REGION Network 51: UNIT 01 STATION 3 COAXIAL HIGH NUMBER OF DEAD PIXELS ALARM
   RUNG wire#powerrail
      { S7_Templates := "SrcType := Int" } EQ_Contact(in1 := "DB16002_U01_STA3_COAXIAL_CLIENT_INTERFACE".U1_STA3_CAM_Read.Variable.Status, in2 := -1)
      Contact( "DB16002_U01_STA3_COAXIAL_CLIENT_INTERFACE".U1_STA3_CAM_Read.Variable.FailedToConnectToCamera )
      wire#w1
      Contact( "DB7254_UNIT_01_STA_3_COAXIAL_ENABLE_DISABLE".ENABLED )
      wire#w2
      Coil( "DB16000_OPC_UA_TRIGGER_ALARM".CLIENT.U1_STA3_COAXIAL.ALARMS.HIGH_NUM_DEAD_PIXELS_A )
   END_RUNG
   RUNG wire#powerrail
      Contact( "DB16000_OPC_UA_TRIGGER_ALARM".CLIENT.U1_STA3_COAXIAL.ALARMS.HIGH_NUM_DEAD_PIXELS_A )
      I_Contact( "DB2120_MPP_ITC_IPC".RESET_FAULTS )
   END_RUNG wire#w1
   RUNG wire#w2
      Coil( "DB426_ALARMS_WARNINGS".UNIT_01.STATION_3_COAXIAL."716645" )
   END_RUNG
   // the same network as SCL:
   "DB16000_OPC_UA_TRIGGER_ALARM".CLIENT.U1_STA3_COAXIAL.ALARMS.HIGH_NUM_DEAD_PIXELS_A := ((("DB16002_U01_STA3_COAXIAL_CLIENT_INTERFACE".U1_STA3_CAM_Read.Variable.Status = (-1)) AND "DB16002_U01_STA3_COAXIAL_CLIENT_INTERFACE".U1_STA3_CAM_Read.Variable.FailedToConnectToCamera) OR ("DB16000_OPC_UA_TRIGGER_ALARM".CLIENT.U1_STA3_COAXIAL.ALARMS.HIGH_NUM_DEAD_PIXELS_A AND NOT "DB2120_MPP_ITC_IPC".RESET_FAULTS)) AND "DB7254_UNIT_01_STA_3_COAXIAL_ENABLE_DISABLE".ENABLED;
   "DB426_ALARMS_WARNINGS".UNIT_01.STATION_3_COAXIAL."716645" := "DB16000_OPC_UA_TRIGGER_ALARM".CLIENT.U1_STA3_COAXIAL.ALARMS.HIGH_NUM_DEAD_PIXELS_A;
END_REGION

REGION Network 52: UNIT 01 STATION 3 COAXIAL CAMERA NO LIGHT DETECTED ALARM
   RUNG wire#powerrail
      { S7_Templates := "SrcType := Int" } EQ_Contact(in1 := "DB16002_U01_STA3_COAXIAL_CLIENT_INTERFACE".U1_STA3_CAM_Read.Variable.Status, in2 := -1)
      Contact( "DB16002_U01_STA3_COAXIAL_CLIENT_INTERFACE".U1_STA3_CAM_Read.Variable.FailedToSetCameraParameters )
      wire#w1
      Contact( "DB7254_UNIT_01_STA_3_COAXIAL_ENABLE_DISABLE".ENABLED )
      wire#w2
      Coil( "DB16000_OPC_UA_TRIGGER_ALARM".CLIENT.U1_STA3_COAXIAL.ALARMS.CAM_NO_LIGHT_DETECTED_A )
   END_RUNG
   RUNG wire#powerrail
      Contact( "DB16000_OPC_UA_TRIGGER_ALARM".CLIENT.U1_STA3_COAXIAL.ALARMS.CAM_NO_LIGHT_DETECTED_A )
      I_Contact( "DB2120_MPP_ITC_IPC".RESET_FAULTS )
   END_RUNG wire#w1
   RUNG wire#w2
      Coil( "DB426_ALARMS_WARNINGS".UNIT_01.STATION_3_COAXIAL."716646" )
   END_RUNG
   // the same network as SCL:
   "DB16000_OPC_UA_TRIGGER_ALARM".CLIENT.U1_STA3_COAXIAL.ALARMS.CAM_NO_LIGHT_DETECTED_A := ((("DB16002_U01_STA3_COAXIAL_CLIENT_INTERFACE".U1_STA3_CAM_Read.Variable.Status = (-1)) AND "DB16002_U01_STA3_COAXIAL_CLIENT_INTERFACE".U1_STA3_CAM_Read.Variable.FailedToSetCameraParameters) OR ("DB16000_OPC_UA_TRIGGER_ALARM".CLIENT.U1_STA3_COAXIAL.ALARMS.CAM_NO_LIGHT_DETECTED_A AND NOT "DB2120_MPP_ITC_IPC".RESET_FAULTS)) AND "DB7254_UNIT_01_STA_3_COAXIAL_ENABLE_DISABLE".ENABLED;
   "DB426_ALARMS_WARNINGS".UNIT_01.STATION_3_COAXIAL."716646" := "DB16000_OPC_UA_TRIGGER_ALARM".CLIENT.U1_STA3_COAXIAL.ALARMS.CAM_NO_LIGHT_DETECTED_A;
END_REGION

REGION Network 53: UNIT 01 STATION 3 COAXIAL CAMERA NO LASER DETECTED ALARM
   RUNG wire#powerrail
      { S7_Templates := "SrcType := Int" } EQ_Contact(in1 := "DB16002_U01_STA3_COAXIAL_CLIENT_INTERFACE".U1_STA3_CAM_Read.Variable.Status, in2 := -1)
      Contact( "DB16002_U01_STA3_COAXIAL_CLIENT_INTERFACE".U1_STA3_CAM_Read.Variable.FailedToSetCameraParameters )
      wire#w1
      Contact( "DB7254_UNIT_01_STA_3_COAXIAL_ENABLE_DISABLE".ENABLED )
      wire#w2
      Coil( "DB16000_OPC_UA_TRIGGER_ALARM".CLIENT.U1_STA3_COAXIAL.ALARMS.CAM_NO_LASER_DETECTED_A )
   END_RUNG
   RUNG wire#powerrail
      Contact( "DB16000_OPC_UA_TRIGGER_ALARM".CLIENT.U1_STA3_COAXIAL.ALARMS.CAM_NO_LASER_DETECTED_A )
      I_Contact( "DB2120_MPP_ITC_IPC".RESET_FAULTS )
   END_RUNG wire#w1
   RUNG wire#w2
      Coil( "DB426_ALARMS_WARNINGS".UNIT_01.STATION_3_COAXIAL."716647" )
   END_RUNG
   // the same network as SCL:
   "DB16000_OPC_UA_TRIGGER_ALARM".CLIENT.U1_STA3_COAXIAL.ALARMS.CAM_NO_LASER_DETECTED_A := ((("DB16002_U01_STA3_COAXIAL_CLIENT_INTERFACE".U1_STA3_CAM_Read.Variable.Status = (-1)) AND "DB16002_U01_STA3_COAXIAL_CLIENT_INTERFACE".U1_STA3_CAM_Read.Variable.FailedToSetCameraParameters) OR ("DB16000_OPC_UA_TRIGGER_ALARM".CLIENT.U1_STA3_COAXIAL.ALARMS.CAM_NO_LASER_DETECTED_A AND NOT "DB2120_MPP_ITC_IPC".RESET_FAULTS)) AND "DB7254_UNIT_01_STA_3_COAXIAL_ENABLE_DISABLE".ENABLED;
   "DB426_ALARMS_WARNINGS".UNIT_01.STATION_3_COAXIAL."716647" := "DB16000_OPC_UA_TRIGGER_ALARM".CLIENT.U1_STA3_COAXIAL.ALARMS.CAM_NO_LASER_DETECTED_A;
END_REGION

REGION Network 54: UNIT 01 STATION 3 COAXIAL CAMERA NO NOZZLE DETECTED ALARM
   RUNG wire#powerrail
      { S7_Templates := "SrcType := Int" } EQ_Contact(in1 := "DB16002_U01_STA3_COAXIAL_CLIENT_INTERFACE".U1_STA3_CAM_Read.Variable.Status, in2 := -1)
      Contact( "DB16002_U01_STA3_COAXIAL_CLIENT_INTERFACE".U1_STA3_CAM_Read.Variable.FailedToSetCameraParameters )
      wire#w1
      Contact( "DB7254_UNIT_01_STA_3_COAXIAL_ENABLE_DISABLE".ENABLED )
      wire#w2
      Coil( "DB16000_OPC_UA_TRIGGER_ALARM".CLIENT.U1_STA3_COAXIAL.ALARMS.CAM_NO_NOZZLE_DETECTED_A )
   END_RUNG
   RUNG wire#powerrail
      Contact( "DB16000_OPC_UA_TRIGGER_ALARM".CLIENT.U1_STA3_COAXIAL.ALARMS.CAM_NO_NOZZLE_DETECTED_A )
      I_Contact( "DB2120_MPP_ITC_IPC".RESET_FAULTS )
   END_RUNG wire#w1
   RUNG wire#w2
      Coil( "DB426_ALARMS_WARNINGS".UNIT_01.STATION_3_COAXIAL."716648" )
   END_RUNG
   // the same network as SCL:
   "DB16000_OPC_UA_TRIGGER_ALARM".CLIENT.U1_STA3_COAXIAL.ALARMS.CAM_NO_NOZZLE_DETECTED_A := ((("DB16002_U01_STA3_COAXIAL_CLIENT_INTERFACE".U1_STA3_CAM_Read.Variable.Status = (-1)) AND "DB16002_U01_STA3_COAXIAL_CLIENT_INTERFACE".U1_STA3_CAM_Read.Variable.FailedToSetCameraParameters) OR ("DB16000_OPC_UA_TRIGGER_ALARM".CLIENT.U1_STA3_COAXIAL.ALARMS.CAM_NO_NOZZLE_DETECTED_A AND NOT "DB2120_MPP_ITC_IPC".RESET_FAULTS)) AND "DB7254_UNIT_01_STA_3_COAXIAL_ENABLE_DISABLE".ENABLED;
   "DB426_ALARMS_WARNINGS".UNIT_01.STATION_3_COAXIAL."716648" := "DB16000_OPC_UA_TRIGGER_ALARM".CLIENT.U1_STA3_COAXIAL.ALARMS.CAM_NO_NOZZLE_DETECTED_A;
END_REGION

REGION Network 55: UNIT 01 STATION 3 COAXIAL CAMERA NO POWDER FLOW DETECTED ALARM
   RUNG wire#powerrail
      { S7_Templates := "SrcType := Int" } EQ_Contact(in1 := "DB16002_U01_STA3_COAXIAL_CLIENT_INTERFACE".U1_STA3_CAM_Read.Variable.Status, in2 := -1)
      Contact( "DB16002_U01_STA3_COAXIAL_CLIENT_INTERFACE".U1_STA3_CAM_Read.Variable.FailedToSetCameraParameters )
      wire#w1
      Contact( "DB7254_UNIT_01_STA_3_COAXIAL_ENABLE_DISABLE".ENABLED )
      wire#w2
      Coil( "DB16000_OPC_UA_TRIGGER_ALARM".CLIENT.U1_STA3_COAXIAL.ALARMS.CAM_NO_POWDER_FLOW_DETECTED_A )
   END_RUNG
   RUNG wire#powerrail
      Contact( "DB16000_OPC_UA_TRIGGER_ALARM".CLIENT.U1_STA3_COAXIAL.ALARMS.CAM_NO_POWDER_FLOW_DETECTED_A )
      I_Contact( "DB2120_MPP_ITC_IPC".RESET_FAULTS )
   END_RUNG wire#w1
   RUNG wire#w2
      Coil( "DB426_ALARMS_WARNINGS".UNIT_01.STATION_3_COAXIAL."716649" )
   END_RUNG
   // the same network as SCL:
   "DB16000_OPC_UA_TRIGGER_ALARM".CLIENT.U1_STA3_COAXIAL.ALARMS.CAM_NO_POWDER_FLOW_DETECTED_A := ((("DB16002_U01_STA3_COAXIAL_CLIENT_INTERFACE".U1_STA3_CAM_Read.Variable.Status = (-1)) AND "DB16002_U01_STA3_COAXIAL_CLIENT_INTERFACE".U1_STA3_CAM_Read.Variable.FailedToSetCameraParameters) OR ("DB16000_OPC_UA_TRIGGER_ALARM".CLIENT.U1_STA3_COAXIAL.ALARMS.CAM_NO_POWDER_FLOW_DETECTED_A AND NOT "DB2120_MPP_ITC_IPC".RESET_FAULTS)) AND "DB7254_UNIT_01_STA_3_COAXIAL_ENABLE_DISABLE".ENABLED;
   "DB426_ALARMS_WARNINGS".UNIT_01.STATION_3_COAXIAL."716649" := "DB16000_OPC_UA_TRIGGER_ALARM".CLIENT.U1_STA3_COAXIAL.ALARMS.CAM_NO_POWDER_FLOW_DETECTED_A;
END_REGION

REGION Network 56: UNIT 1 STATION 3 COAXIAL CAMERA PLC PC MINOR VERSIONS MISMATCH WARNING
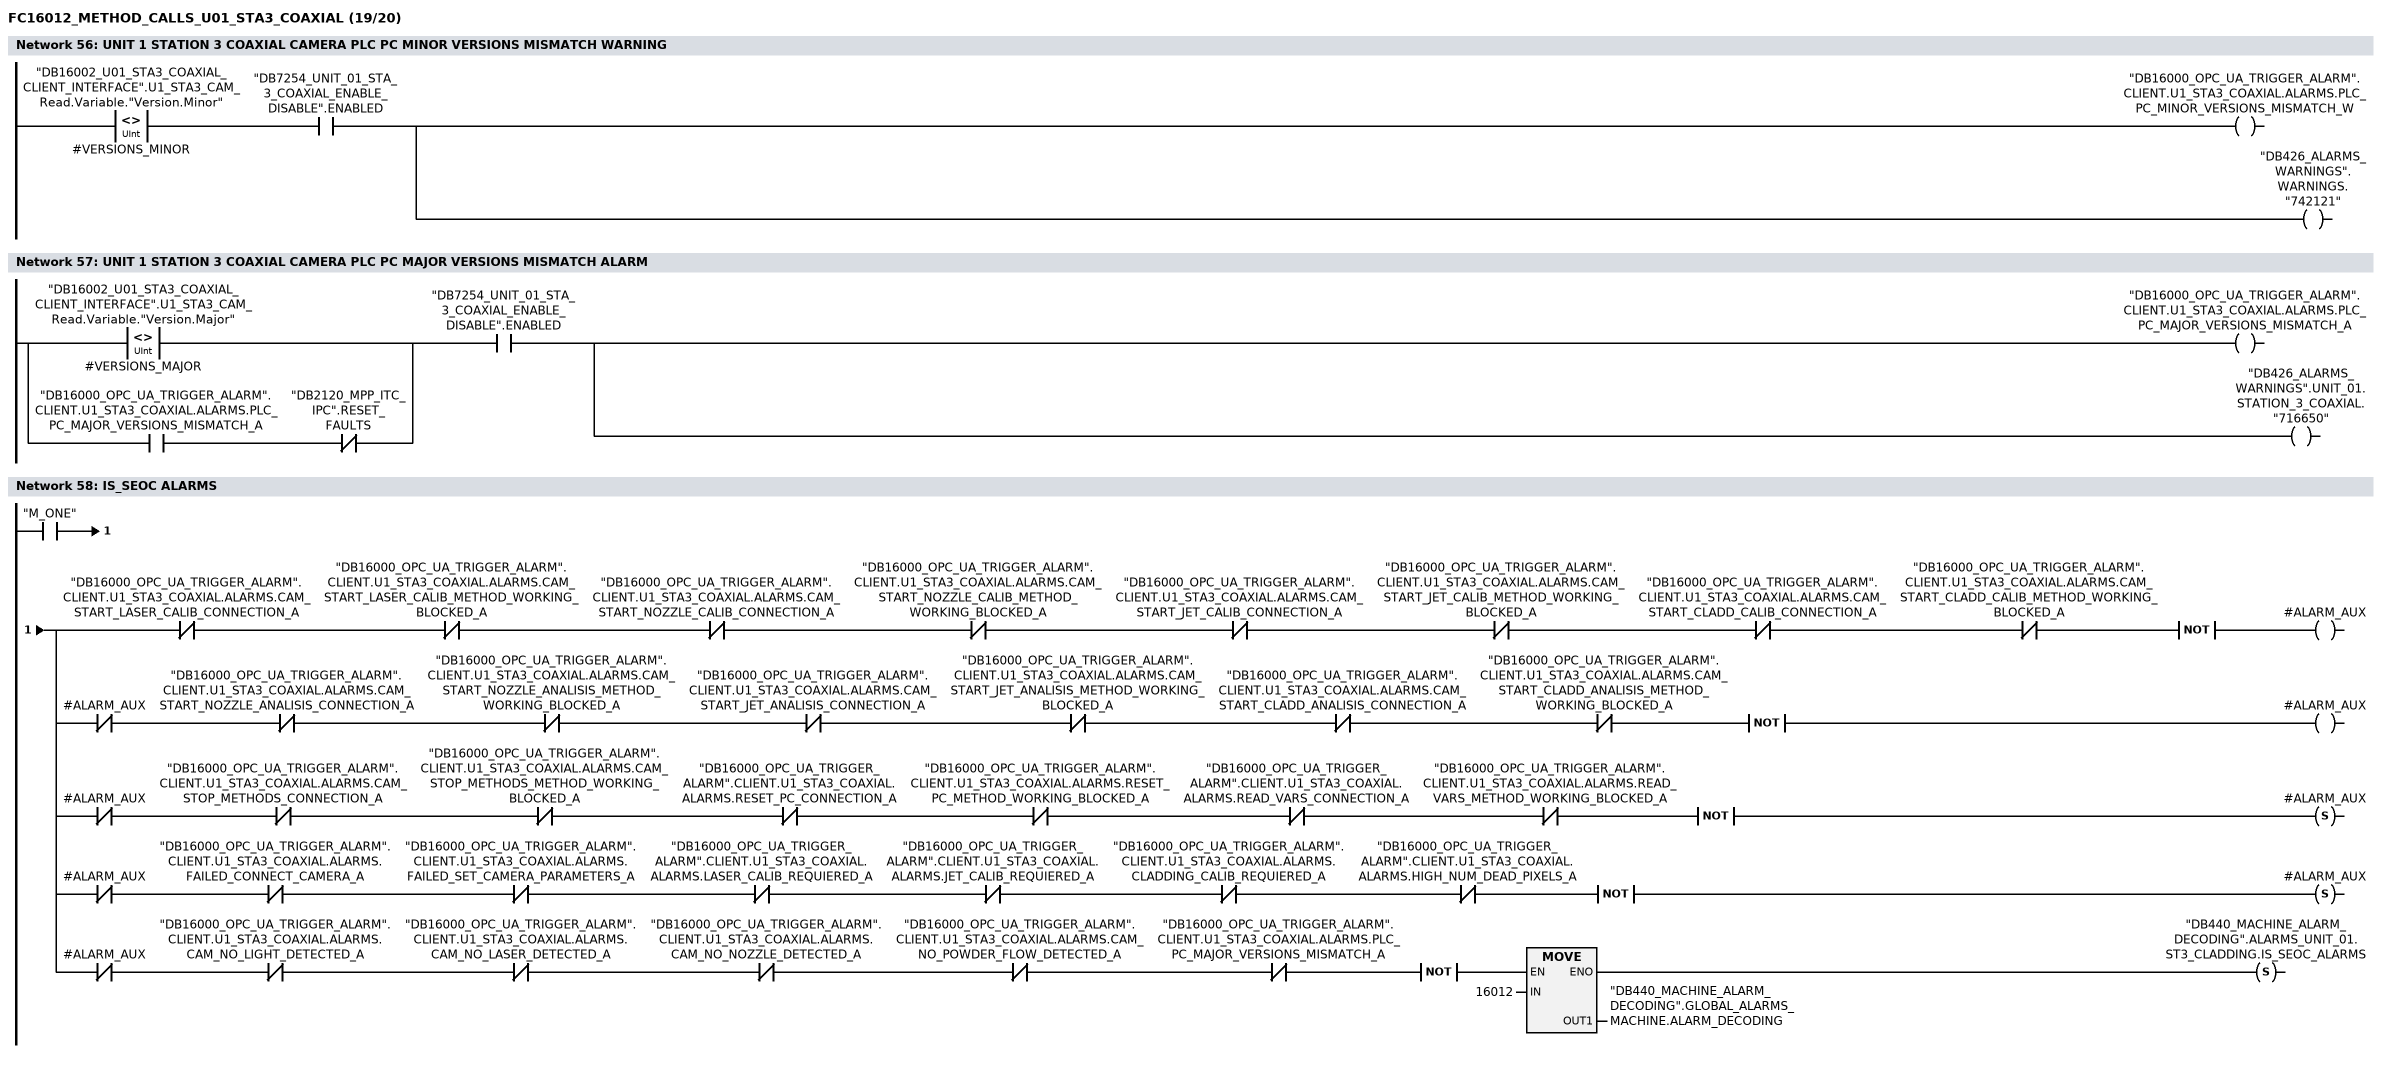
   RUNG wire#powerrail
      { S7_Templates := "SrcType := UInt" } NE_Contact(in1 := "DB16002_U01_STA3_COAXIAL_CLIENT_INTERFACE".U1_STA3_CAM_Read.Variable."Version.Minor", in2 := #VERSIONS_MINOR)
      Contact( "DB7254_UNIT_01_STA_3_COAXIAL_ENABLE_DISABLE".ENABLED )
      wire#w1
      Coil( "DB16000_OPC_UA_TRIGGER_ALARM".CLIENT.U1_STA3_COAXIAL.ALARMS.PLC_PC_MINOR_VERSIONS_MISMATCH_W )
   END_RUNG
   RUNG wire#w1
      Coil( "DB426_ALARMS_WARNINGS".WARNINGS."742121" )
   END_RUNG
   // the same network as SCL:
   "DB16000_OPC_UA_TRIGGER_ALARM".CLIENT.U1_STA3_COAXIAL.ALARMS.PLC_PC_MINOR_VERSIONS_MISMATCH_W := ("DB16002_U01_STA3_COAXIAL_CLIENT_INTERFACE".U1_STA3_CAM_Read.Variable."Version.Minor" <> #VERSIONS_MINOR) AND "DB7254_UNIT_01_STA_3_COAXIAL_ENABLE_DISABLE".ENABLED;
   "DB426_ALARMS_WARNINGS".WARNINGS."742121" := "DB16000_OPC_UA_TRIGGER_ALARM".CLIENT.U1_STA3_COAXIAL.ALARMS.PLC_PC_MINOR_VERSIONS_MISMATCH_W;
END_REGION

REGION Network 57: UNIT 1 STATION 3 COAXIAL CAMERA PLC PC MAJOR VERSIONS MISMATCH ALARM
   RUNG wire#powerrail
      { S7_Templates := "SrcType := UInt" } NE_Contact(in1 := "DB16002_U01_STA3_COAXIAL_CLIENT_INTERFACE".U1_STA3_CAM_Read.Variable."Version.Major", in2 := #VERSIONS_MAJOR)
      wire#w1
      Contact( "DB7254_UNIT_01_STA_3_COAXIAL_ENABLE_DISABLE".ENABLED )
      wire#w2
      Coil( "DB16000_OPC_UA_TRIGGER_ALARM".CLIENT.U1_STA3_COAXIAL.ALARMS.PLC_PC_MAJOR_VERSIONS_MISMATCH_A )
   END_RUNG
   RUNG wire#powerrail
      Contact( "DB16000_OPC_UA_TRIGGER_ALARM".CLIENT.U1_STA3_COAXIAL.ALARMS.PLC_PC_MAJOR_VERSIONS_MISMATCH_A )
      I_Contact( "DB2120_MPP_ITC_IPC".RESET_FAULTS )
   END_RUNG wire#w1
   RUNG wire#w2
      Coil( "DB426_ALARMS_WARNINGS".UNIT_01.STATION_3_COAXIAL."716650" )
   END_RUNG
   // the same network as SCL:
   "DB16000_OPC_UA_TRIGGER_ALARM".CLIENT.U1_STA3_COAXIAL.ALARMS.PLC_PC_MAJOR_VERSIONS_MISMATCH_A := (("DB16002_U01_STA3_COAXIAL_CLIENT_INTERFACE".U1_STA3_CAM_Read.Variable."Version.Major" <> #VERSIONS_MAJOR) OR ("DB16000_OPC_UA_TRIGGER_ALARM".CLIENT.U1_STA3_COAXIAL.ALARMS.PLC_PC_MAJOR_VERSIONS_MISMATCH_A AND NOT "DB2120_MPP_ITC_IPC".RESET_FAULTS)) AND "DB7254_UNIT_01_STA_3_COAXIAL_ENABLE_DISABLE".ENABLED;
   "DB426_ALARMS_WARNINGS".UNIT_01.STATION_3_COAXIAL."716650" := "DB16000_OPC_UA_TRIGGER_ALARM".CLIENT.U1_STA3_COAXIAL.ALARMS.PLC_PC_MAJOR_VERSIONS_MISMATCH_A;
END_REGION

REGION Network 58: IS_SEOC ALARMS
   RUNG wire#powerrail
      Contact( "M_ONE" )
      wire#w1
      I_Contact( "DB16000_OPC_UA_TRIGGER_ALARM".CLIENT.U1_STA3_COAXIAL.ALARMS.CAM_START_LASER_CALIB_CONNECTION_A )
      I_Contact( "DB16000_OPC_UA_TRIGGER_ALARM".CLIENT.U1_STA3_COAXIAL.ALARMS.CAM_START_LASER_CALIB_METHOD_WORKING_BLOCKED_A )
      I_Contact( "DB16000_OPC_UA_TRIGGER_ALARM".CLIENT.U1_STA3_COAXIAL.ALARMS.CAM_START_NOZZLE_CALIB_CONNECTION_A )
      I_Contact( "DB16000_OPC_UA_TRIGGER_ALARM".CLIENT.U1_STA3_COAXIAL.ALARMS.CAM_START_NOZZLE_CALIB_METHOD_WORKING_BLOCKED_A )
      I_Contact( "DB16000_OPC_UA_TRIGGER_ALARM".CLIENT.U1_STA3_COAXIAL.ALARMS.CAM_START_JET_CALIB_CONNECTION_A )
      I_Contact( "DB16000_OPC_UA_TRIGGER_ALARM".CLIENT.U1_STA3_COAXIAL.ALARMS.CAM_START_JET_CALIB_METHOD_WORKING_BLOCKED_A )
      I_Contact( "DB16000_OPC_UA_TRIGGER_ALARM".CLIENT.U1_STA3_COAXIAL.ALARMS.CAM_START_CLADD_CALIB_CONNECTION_A )
      I_Contact( "DB16000_OPC_UA_TRIGGER_ALARM".CLIENT.U1_STA3_COAXIAL.ALARMS.CAM_START_CLADD_CALIB_METHOD_WORKING_BLOCKED_A )
      Not()
      Coil( #ALARM_AUX )
   END_RUNG
   RUNG wire#w1
      I_Contact( #ALARM_AUX )
      I_Contact( "DB16000_OPC_UA_TRIGGER_ALARM".CLIENT.U1_STA3_COAXIAL.ALARMS.CAM_START_NOZZLE_ANALISIS_CONNECTION_A )
      I_Contact( "DB16000_OPC_UA_TRIGGER_ALARM".CLIENT.U1_STA3_COAXIAL.ALARMS.CAM_START_NOZZLE_ANALISIS_METHOD_WORKING_BLOCKED_A )
      I_Contact( "DB16000_OPC_UA_TRIGGER_ALARM".CLIENT.U1_STA3_COAXIAL.ALARMS.CAM_START_JET_ANALISIS_CONNECTION_A )
      I_Contact( "DB16000_OPC_UA_TRIGGER_ALARM".CLIENT.U1_STA3_COAXIAL.ALARMS.CAM_START_JET_ANALISIS_METHOD_WORKING_BLOCKED_A )
      I_Contact( "DB16000_OPC_UA_TRIGGER_ALARM".CLIENT.U1_STA3_COAXIAL.ALARMS.CAM_START_CLADD_ANALISIS_CONNECTION_A )
      I_Contact( "DB16000_OPC_UA_TRIGGER_ALARM".CLIENT.U1_STA3_COAXIAL.ALARMS.CAM_START_CLADD_ANALISIS_METHOD_WORKING_BLOCKED_A )
      Not()
      Coil( #ALARM_AUX )
   END_RUNG
   RUNG wire#w1
      I_Contact( #ALARM_AUX )
      I_Contact( "DB16000_OPC_UA_TRIGGER_ALARM".CLIENT.U1_STA3_COAXIAL.ALARMS.CAM_STOP_METHODS_CONNECTION_A )
      I_Contact( "DB16000_OPC_UA_TRIGGER_ALARM".CLIENT.U1_STA3_COAXIAL.ALARMS.CAM_STOP_METHODS_METHOD_WORKING_BLOCKED_A )
      I_Contact( "DB16000_OPC_UA_TRIGGER_ALARM".CLIENT.U1_STA3_COAXIAL.ALARMS.RESET_PC_CONNECTION_A )
      I_Contact( "DB16000_OPC_UA_TRIGGER_ALARM".CLIENT.U1_STA3_COAXIAL.ALARMS.RESET_PC_METHOD_WORKING_BLOCKED_A )
      I_Contact( "DB16000_OPC_UA_TRIGGER_ALARM".CLIENT.U1_STA3_COAXIAL.ALARMS.READ_VARS_CONNECTION_A )
      I_Contact( "DB16000_OPC_UA_TRIGGER_ALARM".CLIENT.U1_STA3_COAXIAL.ALARMS.READ_VARS_METHOD_WORKING_BLOCKED_A )
      Not()
      S_Coil( #ALARM_AUX )
   END_RUNG
   RUNG wire#w1
      I_Contact( #ALARM_AUX )
      I_Contact( "DB16000_OPC_UA_TRIGGER_ALARM".CLIENT.U1_STA3_COAXIAL.ALARMS.FAILED_CONNECT_CAMERA_A )
      I_Contact( "DB16000_OPC_UA_TRIGGER_ALARM".CLIENT.U1_STA3_COAXIAL.ALARMS.FAILED_SET_CAMERA_PARAMETERS_A )
      I_Contact( "DB16000_OPC_UA_TRIGGER_ALARM".CLIENT.U1_STA3_COAXIAL.ALARMS.LASER_CALIB_REQUIERED_A )
      I_Contact( "DB16000_OPC_UA_TRIGGER_ALARM".CLIENT.U1_STA3_COAXIAL.ALARMS.JET_CALIB_REQUIERED_A )
      I_Contact( "DB16000_OPC_UA_TRIGGER_ALARM".CLIENT.U1_STA3_COAXIAL.ALARMS.CLADDING_CALIB_REQUIERED_A )
      I_Contact( "DB16000_OPC_UA_TRIGGER_ALARM".CLIENT.U1_STA3_COAXIAL.ALARMS.HIGH_NUM_DEAD_PIXELS_A )
      Not()
      S_Coil( #ALARM_AUX )
   END_RUNG
   RUNG wire#w1
      I_Contact( #ALARM_AUX )
      I_Contact( "DB16000_OPC_UA_TRIGGER_ALARM".CLIENT.U1_STA3_COAXIAL.ALARMS.CAM_NO_LIGHT_DETECTED_A )
      I_Contact( "DB16000_OPC_UA_TRIGGER_ALARM".CLIENT.U1_STA3_COAXIAL.ALARMS.CAM_NO_LASER_DETECTED_A )
      I_Contact( "DB16000_OPC_UA_TRIGGER_ALARM".CLIENT.U1_STA3_COAXIAL.ALARMS.CAM_NO_NOZZLE_DETECTED_A )
      I_Contact( "DB16000_OPC_UA_TRIGGER_ALARM".CLIENT.U1_STA3_COAXIAL.ALARMS.CAM_NO_POWDER_FLOW_DETECTED_A )
      I_Contact( "DB16000_OPC_UA_TRIGGER_ALARM".CLIENT.U1_STA3_COAXIAL.ALARMS.PLC_PC_MAJOR_VERSIONS_MISMATCH_A )
      Not()
      Move(in := 16012, out1 => "DB440_MACHINE_ALARM_DECODING".GLOBAL_ALARMS_MACHINE.ALARM_DECODING)
      S_Coil( "DB440_MACHINE_ALARM_DECODING".ALARMS_UNIT_01.ST3_CLADDING.IS_SEOC_ALARMS )
   END_RUNG
   // the same network as SCL:
   #ALARM_AUX := NOT ("M_ONE" AND NOT "DB16000_OPC_UA_TRIGGER_ALARM".CLIENT.U1_STA3_COAXIAL.ALARMS.CAM_START_LASER_CALIB_CONNECTION_A AND NOT "DB16000_OPC_UA_TRIGGER_ALARM".CLIENT.U1_STA3_COAXIAL.ALARMS.CAM_START_LASER_CALIB_METHOD_WORKING_BLOCKED_A AND NOT "DB16000_OPC_UA_TRIGGER_ALARM".CLIENT.U1_STA3_COAXIAL.ALARMS.CAM_START_NOZZLE_CALIB_CONNECTION_A AND NOT "DB16000_OPC_UA_TRIGGER_ALARM".CLIENT.U1_STA3_COAXIAL.ALARMS.CAM_START_NOZZLE_CALIB_METHOD_WORKING_BLOCKED_A AND NOT "DB16000_OPC_UA_TRIGGER_ALARM".CLIENT.U1_STA3_COAXIAL.ALARMS.CAM_START_JET_CALIB_CONNECTION_A AND NOT "DB16000_OPC_UA_TRIGGER_ALARM".CLIENT.U1_STA3_COAXIAL.ALARMS.CAM_START_JET_CALIB_METHOD_WORKING_BLOCKED_A AND NOT "DB16000_OPC_UA_TRIGGER_ALARM".CLIENT.U1_STA3_COAXIAL.ALARMS.CAM_START_CLADD_CALIB_CONNECTION_A AND NOT "DB16000_OPC_UA_TRIGGER_ALARM".CLIENT.U1_STA3_COAXIAL.ALARMS.CAM_START_CLADD_CALIB_METHOD_WORKING_BLOCKED_A);
   #ALARM_AUX := NOT ("M_ONE" AND NOT #ALARM_AUX AND NOT "DB16000_OPC_UA_TRIGGER_ALARM".CLIENT.U1_STA3_COAXIAL.ALARMS.CAM_START_NOZZLE_ANALISIS_CONNECTION_A AND NOT "DB16000_OPC_UA_TRIGGER_ALARM".CLIENT.U1_STA3_COAXIAL.ALARMS.CAM_START_NOZZLE_ANALISIS_METHOD_WORKING_BLOCKED_A AND NOT "DB16000_OPC_UA_TRIGGER_ALARM".CLIENT.U1_STA3_COAXIAL.ALARMS.CAM_START_JET_ANALISIS_CONNECTION_A AND NOT "DB16000_OPC_UA_TRIGGER_ALARM".CLIENT.U1_STA3_COAXIAL.ALARMS.CAM_START_JET_ANALISIS_METHOD_WORKING_BLOCKED_A AND NOT "DB16000_OPC_UA_TRIGGER_ALARM".CLIENT.U1_STA3_COAXIAL.ALARMS.CAM_START_CLADD_ANALISIS_CONNECTION_A AND NOT "DB16000_OPC_UA_TRIGGER_ALARM".CLIENT.U1_STA3_COAXIAL.ALARMS.CAM_START_CLADD_ANALISIS_METHOD_WORKING_BLOCKED_A);
   IF NOT ("M_ONE" AND NOT #ALARM_AUX AND NOT "DB16000_OPC_UA_TRIGGER_ALARM".CLIENT.U1_STA3_COAXIAL.ALARMS.CAM_STOP_METHODS_CONNECTION_A AND NOT "DB16000_OPC_UA_TRIGGER_ALARM".CLIENT.U1_STA3_COAXIAL.ALARMS.CAM_STOP_METHODS_METHOD_WORKING_BLOCKED_A AND NOT "DB16000_OPC_UA_TRIGGER_ALARM".CLIENT.U1_STA3_COAXIAL.ALARMS.RESET_PC_CONNECTION_A AND NOT "DB16000_OPC_UA_TRIGGER_ALARM".CLIENT.U1_STA3_COAXIAL.ALARMS.RESET_PC_METHOD_WORKING_BLOCKED_A AND NOT "DB16000_OPC_UA_TRIGGER_ALARM".CLIENT.U1_STA3_COAXIAL.ALARMS.READ_VARS_CONNECTION_A AND NOT "DB16000_OPC_UA_TRIGGER_ALARM".CLIENT.U1_STA3_COAXIAL.ALARMS.READ_VARS_METHOD_WORKING_BLOCKED_A) THEN
       #ALARM_AUX := TRUE;
   END_IF;
   IF NOT ("M_ONE" AND NOT #ALARM_AUX AND NOT "DB16000_OPC_UA_TRIGGER_ALARM".CLIENT.U1_STA3_COAXIAL.ALARMS.FAILED_CONNECT_CAMERA_A AND NOT "DB16000_OPC_UA_TRIGGER_ALARM".CLIENT.U1_STA3_COAXIAL.ALARMS.FAILED_SET_CAMERA_PARAMETERS_A AND NOT "DB16000_OPC_UA_TRIGGER_ALARM".CLIENT.U1_STA3_COAXIAL.ALARMS.LASER_CALIB_REQUIERED_A AND NOT "DB16000_OPC_UA_TRIGGER_ALARM".CLIENT.U1_STA3_COAXIAL.ALARMS.JET_CALIB_REQUIERED_A AND NOT "DB16000_OPC_UA_TRIGGER_ALARM".CLIENT.U1_STA3_COAXIAL.ALARMS.CLADDING_CALIB_REQUIERED_A AND NOT "DB16000_OPC_UA_TRIGGER_ALARM".CLIENT.U1_STA3_COAXIAL.ALARMS.HIGH_NUM_DEAD_PIXELS_A) THEN
       #ALARM_AUX := TRUE;
   END_IF;
   IF NOT ("M_ONE" AND NOT #ALARM_AUX AND NOT "DB16000_OPC_UA_TRIGGER_ALARM".CLIENT.U1_STA3_COAXIAL.ALARMS.CAM_NO_LIGHT_DETECTED_A AND NOT "DB16000_OPC_UA_TRIGGER_ALARM".CLIENT.U1_STA3_COAXIAL.ALARMS.CAM_NO_LASER_DETECTED_A AND NOT "DB16000_OPC_UA_TRIGGER_ALARM".CLIENT.U1_STA3_COAXIAL.ALARMS.CAM_NO_NOZZLE_DETECTED_A AND NOT "DB16000_OPC_UA_TRIGGER_ALARM".CLIENT.U1_STA3_COAXIAL.ALARMS.CAM_NO_POWDER_FLOW_DETECTED_A AND NOT "DB16000_OPC_UA_TRIGGER_ALARM".CLIENT.U1_STA3_COAXIAL.ALARMS.PLC_PC_MAJOR_VERSIONS_MISMATCH_A) THEN
       "DB440_MACHINE_ALARM_DECODING".GLOBAL_ALARMS_MACHINE.ALARM_DECODING := 16012;
       "DB440_MACHINE_ALARM_DECODING".ALARMS_UNIT_01.ST3_CLADDING.IS_SEOC_ALARMS := TRUE;
   END_IF;
END_REGION

REGION Network 59: WARNINGS
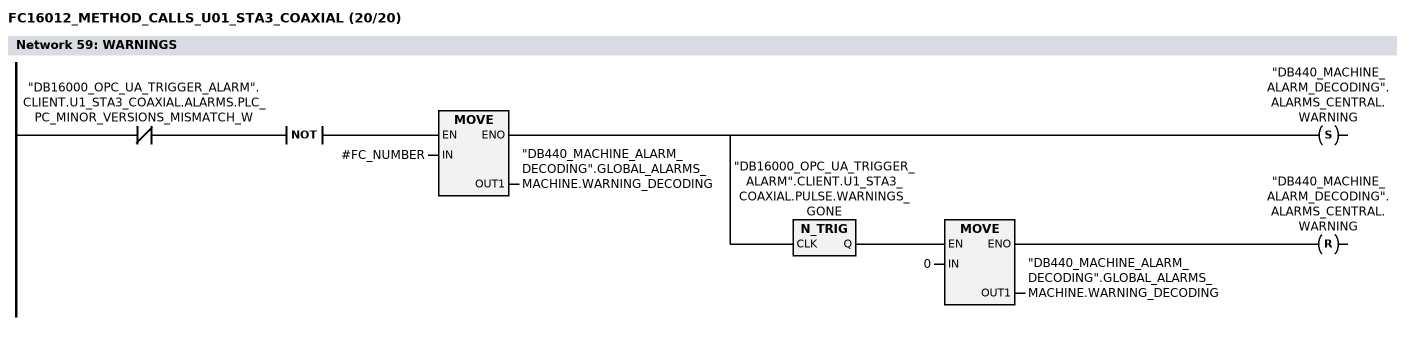
   RUNG wire#powerrail
      I_Contact( "DB16000_OPC_UA_TRIGGER_ALARM".CLIENT.U1_STA3_COAXIAL.ALARMS.PLC_PC_MINOR_VERSIONS_MISMATCH_W )
      Not()
      Move(in := #FC_NUMBER, out1 => "DB440_MACHINE_ALARM_DECODING".GLOBAL_ALARMS_MACHINE.WARNING_DECODING)
      wire#w1
      S_Coil( "DB440_MACHINE_ALARM_DECODING".ALARMS_CENTRAL.WARNING )
   END_RUNG
   RUNG wire#w1
      N_Trig( "DB16000_OPC_UA_TRIGGER_ALARM".CLIENT.U1_STA3_COAXIAL.PULSE.WARNINGS_GONE )
      Move(in := 0, out1 => "DB440_MACHINE_ALARM_DECODING".GLOBAL_ALARMS_MACHINE.WARNING_DECODING)
      R_Coil( "DB440_MACHINE_ALARM_DECODING".ALARMS_CENTRAL.WARNING )
   END_RUNG
   // the same network as SCL:
   #_w1 := NOT (NOT "DB16000_OPC_UA_TRIGGER_ALARM".CLIENT.U1_STA3_COAXIAL.ALARMS.PLC_PC_MINOR_VERSIONS_MISMATCH_W);
   IF #_w1 THEN
       "DB440_MACHINE_ALARM_DECODING".GLOBAL_ALARMS_MACHINE.WARNING_DECODING := #FC_NUMBER;
       "DB440_MACHINE_ALARM_DECODING".ALARMS_CENTRAL.WARNING := TRUE;
   END_IF;
   #_w2 := NOT #_w1 AND "DB16000_OPC_UA_TRIGGER_ALARM".CLIENT.U1_STA3_COAXIAL.PULSE.WARNINGS_GONE;   // falling edge
   "DB16000_OPC_UA_TRIGGER_ALARM".CLIENT.U1_STA3_COAXIAL.PULSE.WARNINGS_GONE := #_w1;
   IF #_w2 THEN
       "DB440_MACHINE_ALARM_DECODING".GLOBAL_ALARMS_MACHINE.WARNING_DECODING := 0;
       "DB440_MACHINE_ALARM_DECODING".ALARMS_CENTRAL.WARNING := FALSE;
   END_IF;
END_REGION
END_FUNCTION
